// TIA Portal project "CicloSR" (V17)

(* hardware
DEVICE "S7-1200 station_1"  S7-1200 Station
   slot 0: "Rack_0"  S7-1200 Rack  Rack  V1.0
   slot 1: "PLC_1"  CPU 1214C AC/DC/Rly  6ES7 214-1BG40-0XB0  V4.5
*)

// ===== PLC "PLC_1"  CPU 1214C AC/DC/Rly =====

VAR_GLOBAL   // PLC tag table "Tabla de variables estándar"
   "Etapa Inicial" AT %M124.0 : Bool;
   "Etapa 1" AT %M124.1 : Bool;
   "Etapa 2" AT %M124.2 : Bool;
   "Etapa 3" AT %M124.3 : Bool;
   "Etapa 4" AT %M124.4 : Bool;
   "System_Byte" AT %MB1 : Byte;
   "FirstScan" AT %M1.0 : Bool;
   "DiagStatusUpdate" AT %M1.1 : Bool;
   "AlwaysTRUE" AT %M1.2 : Bool;
   "AlwaysFALSE" AT %M1.3 : Bool;
   "Clock_Byte" AT %MB0 : Byte;
   "Clock_10Hz" AT %M0.0 : Bool;
   "Clock_5Hz" AT %M0.1 : Bool;
   "Clock_2.5Hz" AT %M0.2 : Bool;
   "Clock_2Hz" AT %M0.3 : Bool;
   "Clock_1.25Hz" AT %M0.4 : Bool;
   "Clock_1Hz" AT %M0.5 : Bool;
   "Clock_0.625Hz" AT %M0.6 : Bool;
   "Clock_0.5Hz" AT %M0.7 : Bool;
   "Tag_6" AT %M14.0 : Bool;
   "Tag_1" AT %M14.4 : Bool;
   "Tag_2" AT %M125.1 : Bool;
   "Tag_3" AT %M215.0 : Bool;
   "Tag_4" AT %M215.1 : Bool;
   "Tag_5" AT %M215.2 : Bool;
   "Tag_7" AT %I124.1 : Bool;
END_VAR

DATA_BLOCK "CicloDatos"   // DB1
{ S7_Optimized_Access := 'TRUE' }
VERSION : 0.1
   VAR
      Start_Cycle : Bool;
      On_cycle : Bool;
      End_Cycle : Bool;
      Aux_1 : Bool;
      Aux_2 : Bool;
      Aux_3 : Bool;
      Aux_4 : Bool;
      Aux_5 : Bool;
      Aux_6 : Bool;
      Aux_7 : Bool;
      Aux_8 : Bool;
      Step_1 : Bool;
      Step_2 : Bool;
      Step_3 : Bool;
      Step_4 : Bool;
      Step_5 : Bool;
      Step_6 : Bool;
      Step_7 : Bool;
      Step_8 : Bool;
   END_VAR
BEGIN
END_DATA_BLOCK

// folder: System blocks/Program resources

DATA_BLOCK "IEC_Counter_0_DB"   // DB2
{ S7_Optimized_Access := 'TRUE' }
AUTHOR : Simatic
FAMILY : IEC
NAME : CNTR
VERSION : 1.0
// stored: InstanceOfName IEC_COUNTER
"IEC_COUNTER"
BEGIN
END_DATA_BLOCK

// folder: (top level)

FUNCTION "Ciclo" : Void   // FC1, LAD
{ S7_Optimized_Access := 'TRUE' }
VERSION : 0.1
   VAR_TEMP   // added for the SCL form of the ladder/FBD networks
      _w1 : Bool;
      _w2 : Bool;
   END_VAR
BEGIN

REGION Network 1
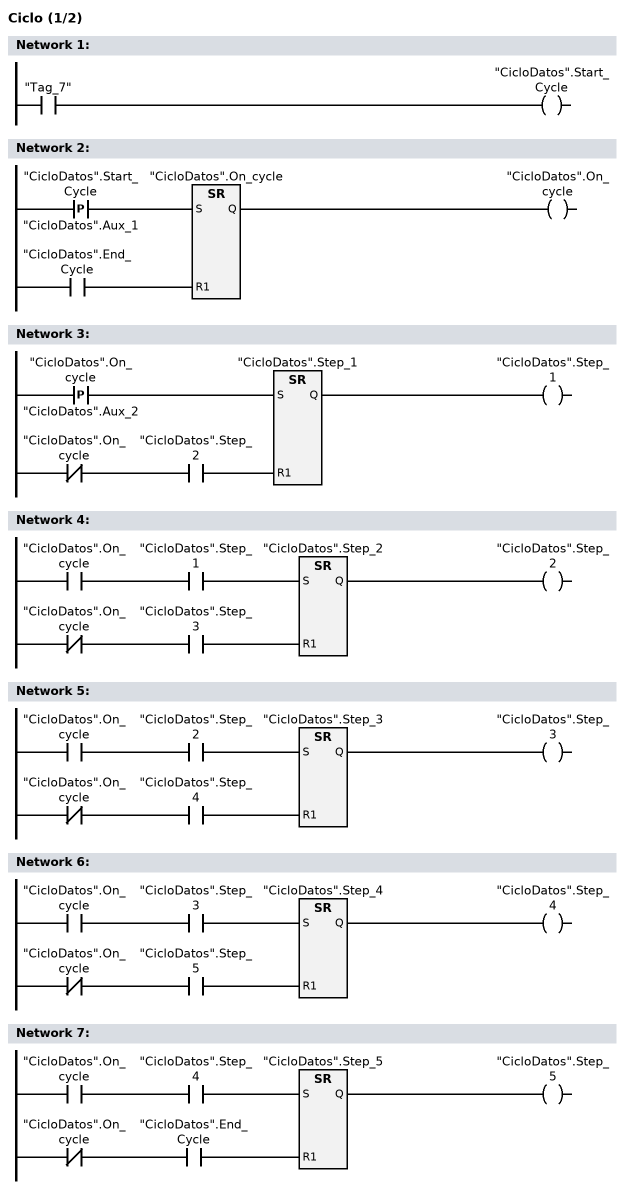
   RUNG wire#powerrail
      Contact( "Tag_7" )
      Coil( "CicloDatos".Start_Cycle )
   END_RUNG
   // the same network as SCL:
   "CicloDatos".Start_Cycle := "Tag_7";
END_REGION

REGION Network 2
   RUNG wire#powerrail
      P_Contact(operand := "CicloDatos".Start_Cycle, bit := "CicloDatos".Aux_1)
      S_SR(operand := "CicloDatos".On_cycle, r1 := wire#w1)
      Coil( "CicloDatos".On_cycle )
   END_RUNG
   RUNG wire#powerrail
      Contact( "CicloDatos".End_Cycle )
   END_RUNG wire#w1
   // the same network as SCL:
   #_w1 := "CicloDatos".Start_Cycle AND NOT "CicloDatos".Aux_1;   // rising edge of "CicloDatos".Start_Cycle
   "CicloDatos".Aux_1 := "CicloDatos".Start_Cycle;
   IF #_w1 THEN
       "CicloDatos".On_cycle := TRUE;   // SR flip-flop
   END_IF;
   IF "CicloDatos".End_Cycle THEN "CicloDatos".On_cycle := FALSE; END_IF;
   "CicloDatos".On_cycle := "CicloDatos".On_cycle;
END_REGION

REGION Network 3
   RUNG wire#powerrail
      P_Contact(operand := "CicloDatos".On_cycle, bit := "CicloDatos".Aux_2)
      S_SR(operand := "CicloDatos".Step_1, r1 := wire#w1)
      Coil( "CicloDatos".Step_1 )
   END_RUNG
   RUNG wire#powerrail
      I_Contact( "CicloDatos".On_cycle )
      Contact( "CicloDatos".Step_2 )
   END_RUNG wire#w1
   // the same network as SCL:
   #_w1 := "CicloDatos".On_cycle AND NOT "CicloDatos".Aux_2;   // rising edge of "CicloDatos".On_cycle
   "CicloDatos".Aux_2 := "CicloDatos".On_cycle;
   IF #_w1 THEN
       "CicloDatos".Step_1 := TRUE;   // SR flip-flop
   END_IF;
   IF NOT "CicloDatos".On_cycle AND "CicloDatos".Step_2 THEN "CicloDatos".Step_1 := FALSE; END_IF;
   "CicloDatos".Step_1 := "CicloDatos".Step_1;
END_REGION

REGION Network 4
   RUNG wire#powerrail
      Contact( "CicloDatos".On_cycle )
      Contact( "CicloDatos".Step_1 )
      S_SR(operand := "CicloDatos".Step_2, r1 := wire#w1)
      Coil( "CicloDatos".Step_2 )
   END_RUNG
   RUNG wire#powerrail
      I_Contact( "CicloDatos".On_cycle )
      Contact( "CicloDatos".Step_3 )
   END_RUNG wire#w1
   // the same network as SCL:
   IF "CicloDatos".On_cycle AND "CicloDatos".Step_1 THEN
       "CicloDatos".Step_2 := TRUE;   // SR flip-flop
   END_IF;
   IF NOT "CicloDatos".On_cycle AND "CicloDatos".Step_3 THEN "CicloDatos".Step_2 := FALSE; END_IF;
   "CicloDatos".Step_2 := "CicloDatos".Step_2;
END_REGION

REGION Network 5
   RUNG wire#powerrail
      Contact( "CicloDatos".On_cycle )
      Contact( "CicloDatos".Step_2 )
      S_SR(operand := "CicloDatos".Step_3, r1 := wire#w1)
      Coil( "CicloDatos".Step_3 )
   END_RUNG
   RUNG wire#powerrail
      I_Contact( "CicloDatos".On_cycle )
      Contact( "CicloDatos".Step_4 )
   END_RUNG wire#w1
   // the same network as SCL:
   IF "CicloDatos".On_cycle AND "CicloDatos".Step_2 THEN
       "CicloDatos".Step_3 := TRUE;   // SR flip-flop
   END_IF;
   IF NOT "CicloDatos".On_cycle AND "CicloDatos".Step_4 THEN "CicloDatos".Step_3 := FALSE; END_IF;
   "CicloDatos".Step_3 := "CicloDatos".Step_3;
END_REGION

REGION Network 6
   RUNG wire#powerrail
      Contact( "CicloDatos".On_cycle )
      Contact( "CicloDatos".Step_3 )
      S_SR(operand := "CicloDatos".Step_4, r1 := wire#w1)
      Coil( "CicloDatos".Step_4 )
   END_RUNG
   RUNG wire#powerrail
      I_Contact( "CicloDatos".On_cycle )
      Contact( "CicloDatos".Step_5 )
   END_RUNG wire#w1
   // the same network as SCL:
   IF "CicloDatos".On_cycle AND "CicloDatos".Step_3 THEN
       "CicloDatos".Step_4 := TRUE;   // SR flip-flop
   END_IF;
   IF NOT "CicloDatos".On_cycle AND "CicloDatos".Step_5 THEN "CicloDatos".Step_4 := FALSE; END_IF;
   "CicloDatos".Step_4 := "CicloDatos".Step_4;
END_REGION

REGION Network 7
   RUNG wire#powerrail
      Contact( "CicloDatos".On_cycle )
      Contact( "CicloDatos".Step_4 )
      S_SR(operand := "CicloDatos".Step_5, r1 := wire#w1)
      Coil( "CicloDatos".Step_5 )
   END_RUNG
   RUNG wire#powerrail
      I_Contact( "CicloDatos".On_cycle )
      Contact( "CicloDatos".End_Cycle )
   END_RUNG wire#w1
   // the same network as SCL:
   IF "CicloDatos".On_cycle AND "CicloDatos".Step_4 THEN
       "CicloDatos".Step_5 := TRUE;   // SR flip-flop
   END_IF;
   IF NOT "CicloDatos".On_cycle AND "CicloDatos".End_Cycle THEN "CicloDatos".Step_5 := FALSE; END_IF;
   "CicloDatos".Step_5 := "CicloDatos".Step_5;
END_REGION

REGION Network 8
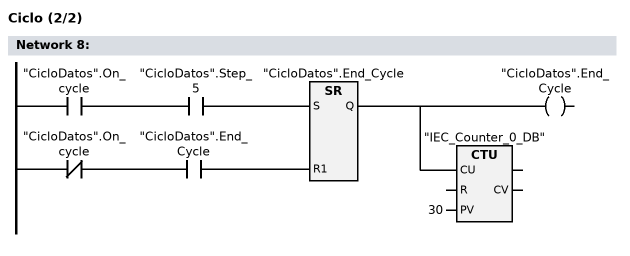
   #_w1 := NOT "CicloDatos".On_cycle AND "CicloDatos".End_Cycle;
   IF "CicloDatos".On_cycle AND "CicloDatos".Step_5 THEN
       "CicloDatos".End_Cycle := TRUE;   // SR flip-flop
   END_IF;
   IF #_w1 THEN "CicloDatos".End_Cycle := FALSE; END_IF;
   #_w2 := "CicloDatos".End_Cycle;
   "CicloDatos".End_Cycle := "CicloDatos".End_Cycle;
   "IEC_Counter_0_DB".CTU(CU := #_w2, PV := 30);
END_REGION
END_FUNCTION

ORGANIZATION_BLOCK "Main"   // OB1, LAD, ProgramCycle
TITLE = "Main Program Sweep (Cycle)"
{ S7_Optimized_Access := 'TRUE' }
VERSION : 0.1
   VAR_INPUT
      Initial_Call : Bool;   // Initial call of this OB
      Remanence : Bool;   // =True, if remanent data are available
   END_VAR
BEGIN

REGION Network 1
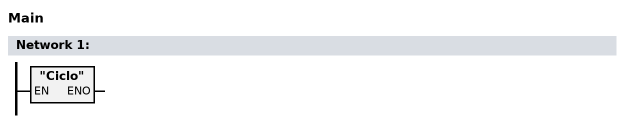
   RUNG wire#powerrail
      "Ciclo"()
   END_RUNG
   // the same network as SCL:
   "Ciclo"();
END_REGION
END_ORGANIZATION_BLOCK